TYPE AX5000_P_0602 :
STRUCT
	Predictive_torque_command_value:INT;
END_STRUCT
END_TYPE

(* stored: Version 1.1.0.1, ProductVersion 3.1.4024.3
   DUT AX5000_P_0602: Id {72d60779-5f35-4a6d-841e-99c8a1fd582c} *)
